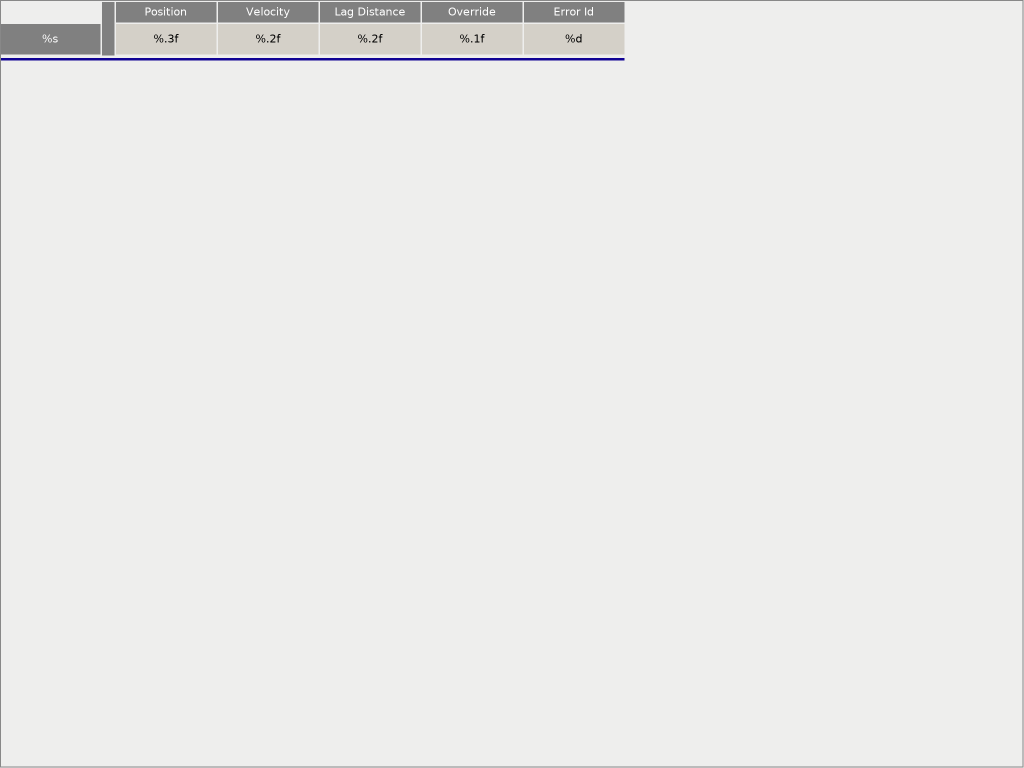
VISUALIZATION VisuAxisInfo  // 1024x768
VAR_IN_OUT
	sAxisName		: STRING;
	stAxisRefVisu	: AXIS_REF;
END_VAR
    Rectangle (0,24 100x30), "%s", text variable: sAxisName
    Rectangle (116,24 100x30), "%.3f", text variable: stAxisRefVisu.NcToPlc.ActPos
    Rectangle (116,2 100x20), "Position"
    Rectangle (218,24 100x30), "%.2f", text variable: stAxisRefVisu.NcToPlc.ActVelo
    Rectangle (422,24 100x30), "%.1f", text variable: stAxisRefVisu.PlcToNc.Override / 10000
    Rectangle (218,2 100x20), "Velocity"
    Rectangle (422,2 100x20), "Override"
    Rectangle (524,24 100x30), "%d", text variable: stAxisRefVisu.Status.ErrorID
    Rectangle (524,2 100x20), "Error Id"
    Rectangle (320,24 100x30), "%.2f", text variable: stAxisRefVisu.NcToPlc.PosDiff
    Rectangle (320,2 100x20), "Lag Distance"
    RoundedRectangle (102,2 12x53), colour toggle: stAxisRefVisu.Status.ControlLoopClosed
    RoundedRectangle (0,58 624x2)
END_VISUALIZATION

(* stored: Version 1.1.0.1, ProductVersion 3.1.4022.6
   Visu VisuAxisInfo: Id {27603c2b-9445-4e38-8d5c-973ea176b2c5} *)
